{attribute 'qualified_only'}
{attribute 'strict'}
{attribute 'to_string'}
TYPE E_DS402EGU :
(
    MM:=0,
    UM:=1,
    NM:=2
);
END_TYPE

(* stored: Version 1.1.0.1
   DUT E_DS402EGU: Id {2b79b46c-17fb-44ec-a844-3194a4ea453a} *)
